# B&R Automation Studio project DeltaTracking (part 2)

#### Cyclic.st - Cyclic code
```iecst
PROGRAM _CYCLIC
	DefineLinks;

	CASE State OF

		/////////////////////////////////////////////////////////////////////////////
		STATE_WAIT:
			/////////////////////////////////////////////////////////////////////////////
			IF  Start THEN
				State := 	STATE_INIT;
			END_IF

		/////////////////////////////////////////////////////////////////////////////
		STATE_INIT:
		////////////////////////////////////////////////////////////////////////////

			IF MpAxConveyor.CommandBusy THEN
				// wait
			ELSIF 	NOT(MpAxConveyor.Active) THEN
				MpAxConveyor.Enable := TRUE;

			ELSIF MpAxConveyor.Error THEN
				MpAxConveyor.ErrorReset := TRUE;

			ELSIF NOT(MpAxConveyor.PowerOn) THEN
				MpAxConveyor.Power := TRUE;

			ELSIF NOT(MpAxConveyor.IsHomed) THEN
				AxParConveyor.Homing.Mode := mcHOMING_DIRECT;
				AxParConveyor.Homing.Position := 0;
				MpAxConveyor.Home := TRUE;

			ELSIF MpAxConveyor.Info.CommunicationReady THEN
				LastProductPosition := MpAxConveyor.Position - ProductGap;
				MC_BR_TrackingFrameDelete_0.Execute := TRUE;
				State := STATE_PRODUCTION;
			END_IF

		//////////////////////////////////////// Frame Handling! + Stat Machine Conveyor///////////////////////////////////////
		STATE_PRODUCTION:
		///////////////////////////////////////////////////////////////////////////////////////////////////////////////////////

			// Move Belt with selected speed
			IF AxParConveyor.Velocity  <> SetVelocity THEN
				// If velocity ist not up to date, update Conveyer Velocity to the Velocity set at the ControlPanel
				MpAxConveyor.Update := TRUE;
			END_IF
			AxParConveyor.Velocity := SetVelocity;
			MpAxConveyor.MoveVelocity := TRUE;

			IF NOT MC_BR_TrackingFrameCreate_0.Busy THEN
				addNewObjects;
			END_IF

			IF MpAxConveyor.Error THEN
				State := STATE_ERROR;

			ELSIF NOT Start THEN
				MpAxConveyor.MoveVelocity := FALSE;

				IF (MpAxConveyor.Error) THEN
					MpAxConveyor.Power := FALSE;
					State := STATE_WAIT;

				ELSIF MpAxConveyor.PowerOn AND NOT(MpAxConveyor.CommandBusy) THEN
					MpAxConveyor.MoveVelocity := FALSE;
					MpAxConveyor.Power := FALSE;

				ELSIF NOT(MpAxConveyor.CommandBusy) THEN
					State := STATE_WAIT;

				END_IF
			END_IF

		///////////////////////////////////////////////////////////////////////////////
		STATE_ERROR:
		///////////////////////////////////////////////////////////////////////////////
			MpAxConveyor.MoveVelocity := FALSE;
			MpAxConveyor.Power := FALSE;

			IF Reset AND MpAxConveyor.Error AND MpAxConveyor.CommandBusy THEN
				MpAxConveyor.ErrorReset := TRUE;

			ELSIF Start AND NOT(MpAxConveyor.Error) AND NOT(MpAxConveyor.CommandBusy) THEN
				State := STATE_WAIT;
			END_IF

	END_CASE

	MpAxConveyor(MpLink := LinkAxis, Parameters := ADR(AxParConveyor), ErrorReset := Reset);
	MC_BR_TrackingFrameCreate_0(TrackingPath := LinkTrackingPath);
	MC_BR_TrackingFrameDelete_0(TrackingPath := LinkTrackingPath);

	IF (MpAxConveyor.Update AND MpAxConveyor.UpdateDone) OR MpAxConveyor.Error THEN
		MpAxConveyor.Update	:= FALSE;
	END_IF

	IF (NOT(MpAxConveyor.MoveActive) AND NOT(MpAxConveyor.CommandBusy)) OR MpAxConveyor.Error THEN
		MpAxConveyor.MoveVelocity := FALSE;
		MpAxConveyor.Update := FALSE;
	END_IF

	IF MpAxConveyor.ErrorReset AND NOT(MpAxConveyor.Error) THEN
		MpAxConveyor.ErrorReset := FALSE;
	END_IF

	IF (MpAxConveyor.Home AND MpAxConveyor.IsHomed) OR MpAxConveyor.Error THEN
		MpAxConveyor.Home := FALSE;
	END_IF

	MC_BR_TrackingFrameCreate_0.Execute	:= FALSE;
	MC_BR_TrackingFrameDelete_0.Execute := FALSE;

END_PROGRAM
```

#### Exit.st - Exit code
```iecst
PROGRAM _EXIT

END_PROGRAM
```

#### DeviceActions.st
```iecst
ACTION addNewObjects:

	// overflow handling
	IF MpAxConveyor.Position < LastProductPosition THEN
		LastProductPosition := LastProductPosition - Period;
	END_IF

	IF MpAxConveyor.Position <  LastProductPosition	+ ProductGap THEN
		RETURN;
	END_IF

	IF Multipick THEN
		MC_BR_TrackingFrameCreate_0.Parameters.Translation.Y := 80 - UDINT_TO_LREAL(createCnt MOD 2) * 160;
		createCnt := createCnt + 1;

		IF createCnt MOD 2 = 0 THEN
			LastProductPosition := MpAxConveyor.Position;
		END_IF

	ELSE
		IF RandomCreation THEN
			MC_BR_TrackingFrameCreate_0.Parameters.Translation.Y := (UINT_TO_LREAL((TIM_musec()*10) MOD 160) - 80);
			MC_BR_TrackingFrameCreate_0.Parameters.Orientation.Angle3 := (UINT_TO_LREAL((TIM_musec()*10) MOD 178)-89);
		ELSE
			MC_BR_TrackingFrameCreate_0.Parameters.Translation.Y := 0;
			MC_BR_TrackingFrameCreate_0.Parameters.Orientation.Angle3 := 0;
		END_IF
		LastProductPosition := MpAxConveyor.Position;
	END_IF

	// simulate two diffent product types
	MC_BR_TrackingFrameCreate_0.Parameters.Attribute := 2#0001;
	IF (TIM_ticks() MOD 2) = 1 THEN
		MC_BR_TrackingFrameCreate_0.Parameters.Attribute := 2#0011;
	END_IF;

	// Add frame in the buffer
	MC_BR_TrackingFrameCreate_0.Parameters.LatchedPath.Position := MpAxConveyor.Position;
	MC_BR_TrackingFrameCreate_0.Execute	:= TRUE;

END_ACTION
```

#### DefineLinks.st
```iecst
ACTION DefineLinks:
	LinkTrackingPath := ADR(gTrackingPathConveyor_1);
	LinkAxis := ADR(gAxis_Conveyor_1);
	Period := 100000.0;

	Reset := ControlPanel.Input.Reset;
	Start :=
		(ControlPanel.Input.StartMultipick OR
		ControlPanel.Input.StartPickNPlace OR
		ControlPanel.Input.StartPlaceWithConditionalStop OR
		ControlPanel.Input.StartPrePalletizing OR
		ControlPanel.Input.StartSorting OR
		ControlPanel.Input.StartMultipickRandom);

	Multipick := ControlPanel.Input.StartMultipick;
	ProductGap := ControlPanel.Input.ProductGap;
	SetVelocity := ControlPanel.Input.VelocityProduction;
	RandomCreation := ControlPanel.Input.StartMultipickRandom;

END_ACTION
```

### Program Logical/Conveyor/APP_Conveyor2 (IEC)

- Cyclic.st (reference to Logical/Conveyor/APP_Conveyor1/Cyclic.st)

- DeviceActions.st (reference to Logical/Conveyor/APP_Conveyor1/DeviceActions.st)

- Exit.st (reference to Logical/Conveyor/APP_Conveyor1/Exit.st)

- Init.st (reference to Logical/Conveyor/APP_Conveyor1/Init.st)

- Variables.var (reference to Logical/Conveyor/APP_Conveyor1/Variables.var)

#### DefineLinks.st
```iecst
ACTION DefineLinks:
	LinkTrackingPath := ADR(gTrackingPathConveyor_2);
	LinkAxis := ADR(gAxis_Conveyor_2);
	Period := 100000.0;

	Reset := ControlPanel.Input.Reset;
	Start :=
		(ControlPanel.Input.StartMultipick OR
		ControlPanel.Input.StartPickNPlace OR
		ControlPanel.Input.StartPlaceWithConditionalStop OR
		ControlPanel.Input.StartPrePalletizing OR
		ControlPanel.Input.StartSorting OR
		ControlPanel.Input.StartMultipickRandom);

	Multipick := ControlPanel.Input.StartMultipick;
	ProductGap := ControlPanel.Input.ProductGap;
	SetVelocity := ControlPanel.Input.VelocityProduction;
	RandomCreation := ControlPanel.Input.StartMultipickRandom;

END_ACTION
```

### Robot.typ
```iecst
TYPE
	RobotStatesEnum :
		( (*State of the robot*)
		ROBOT_WAIT,
		ROBOT_RESET,
		ROBOT_POWER,
		ROBOT_HOME,
		ROBOT_MOVE,
		ROBOT_PRODUCTION,
		ROBOT_ERROR
		);
END_TYPE
```

### Program Logical/Robots/APP_Robot1 (IEC) - Delta1

#### CommonVars.var - Local variables
```iecst
(*
Link handling*)
VAR
	NameAxesGroup : STRING[250]; (*Name of axGroup to find position in object hierachy*)
	LinkAxesGroup : UDINT; (*Link to delta*)
	NameTrackingPath : STRING[250];
	LinkAxisTrackingPath : UDINT;
	LinkTrackingPath : UDINT;
END_VAR
(*
Robot Interface Definition*)
VAR
	MC_BR_GroupStop_X : MC_GroupStop; (*Group object to home axis group*)
	MC_BR_GroupHome_X : MC_BR_GroupHome_15; (*Group object to home axis group*)
	MC_GroupReset_X : MC_GroupReset; (*Group object to home axis group*)
	MC_BR_GroupPower_X : MC_BR_GroupPower; (*Group object to home axis group*)
	MC_BR_GroupReadInfo_X : MC_BR_GroupReadInfo; (*Group object to home axis group*)
	MC_BR_MoveProgram_X : MC_BR_MoveProgram; (*Group object to home axis group*)
	MC_BR_ConditionalStop_0 : MC_BR_ConditionalStop;
	MC_BR_TrackingStatus_PathGen_X : MC_BR_TrackingStatus_PathGen;
	MC_BR_PathInfo_0 : MC_BR_PathInfo;
	MC_BR_GroupReadCyclicPosition_X : MC_BR_GroupReadCyclicPosition_15;
END_VAR
(*
Variables used handling objects and reading informations about the robot*)
VAR
	MC_BR_GetCoordSystemIdent_X : MC_BR_GetCoordSystemIdent;
	MC_BR_TrackingFrameCreate_X : MC_BR_TrackingFrameCreate; (*Tracking Path, read all objects on Path*)
	MC_BR_ReadCyclicPosition_X : MC_BR_ReadCyclicPosition; (*Tracking Path, read all objects on Path*)
END_VAR
(*
Logic*)
VAR
	Reset : BOOL;
	Start : BOOL;
	State : RobotStatesEnum; (*Statemachine*)
END_VAR
(*
Scene Viewer*)
VAR
	GripperClosed : BOOL; (*Scene Viewer*)
	MultigripperClosedPos1 : BOOL; (*Scene Viewer*)
	MultigripperClosedPos2 : BOOL; (*Scene Viewer*)
END_VAR
(*
ST Var*)
VAR
	M16 : BOOL; (*ST Var*)
	M17 : BOOL; (*ST Var*)
	M32 : BOOL; (*ST Var*)
	M33 : BOOL; (*ST Var*)
	M34 : BOOL; (*ST Var*)
	M40 : BOOL; (*ST Var*)
END_VAR
(*
Monitorin Elements*)
VAR
	PickRateWaitForSync : BOOL;
	PickRateCount : UDINT;
	PickRateTimestamp : TIME;
	PickRateTrackingPath : REFERENCE TO McTrackingPathType;
	PickRate : LREAL;
END_VAR
```

#### Init.st - Init code
```iecst
PROGRAM _INIT

	// This action defines the links to the conveyeor and the robot
	DefineLinks;

	MC_BR_PathInfo_0.Enable := TRUE;
	MC_BR_GroupReadInfo_X.Enable := TRUE;
	MC_BR_GroupReadCyclicPosition_X.Enable := TRUE;

	MC_BR_ConditionalStop_0.Enable := TRUE;
	MC_BR_ConditionalStop_0.Identifier := 123;
	MC_BR_ConditionalStop_0.Deactivate := TRUE;
	MC_BR_ConditionalStop_0.Reactivate := FALSE;

	MC_BR_GetCoordSystemIdent_X.CoordSystemName := NameTrackingPath;
	MC_BR_GetCoordSystemIdent_X.Execute := TRUE;
	MC_BR_GetCoordSystemIdent_X();

	MC_BR_ReadCyclicPosition_X.Enable := TRUE;
	MC_BR_ReadCyclicPosition_X.ValueSource := mcVALUE_ACTUAL;

	MC_BR_GroupReadCyclicPosition_X.CoordSystem := MC_BR_GetCoordSystemIdent_X.Ident;

	MC_BR_TrackingStatus_PathGen_X.Enable := TRUE;

END_PROGRAM
```

#### Cyclic.st
```iecst
PROGRAM _CYCLIC
	DefineLinks;

	CASE State OF

		/////////////////////////////////////////////////////////////////////////////
		ROBOT_WAIT:
		/////////////////////////////////////////////////////////////////////////////
			IF  Start THEN
				State := ROBOT_RESET;
			END_IF
			MC_BR_GroupPower_X.Enable := FALSE;
			MultigripperClosedPos1 := FALSE;
			MultigripperClosedPos2 := FALSE;
			GripperClosed := FALSE;
			PickRateCount := 0;

		/////////////////////////////////////////////////////////////////////////////
		ROBOT_RESET:
		/////////////////////////////////////////////////////////////////////////////
			MC_GroupReset_X.Execute := TRUE;
			IF MC_GroupReset_X.Done THEN
				State := ROBOT_POWER;
			END_IF

		/////////////////////////////////////////////////////////////////////////////
		ROBOT_POWER:
		/////////////////////////////////////////////////////////////////////////////
			MC_BR_GroupPower_X.Enable := TRUE;
			IF MC_BR_GroupPower_X.Status THEN
				State := ROBOT_HOME;
			END_IF

		/////////////////////////////////////////////////////////////////////////////
		ROBOT_HOME:
		/////////////////////////////////////////////////////////////////////////////
			MC_BR_GroupHome_X.Execute := TRUE;
			IF MC_BR_GroupHome_X.Done THEN
				State := ROBOT_MOVE;
			END_IF

		/////////////////////////////////////////////////////////////////////////////
		ROBOT_MOVE:
		/////////////////////////////////////////////////////////////////////////////
			MC_BR_MoveProgram_X.Execute := TRUE;
			IF MC_BR_MoveProgram_X.Active THEN
				State := ROBOT_PRODUCTION;
			END_IF

		/////////////////////////////////////////////////////////////////////////////
		ROBOT_PRODUCTION:
		/////////////////////////////////////////////////////////////////////////////

			operateGripper;
			updateConditionalStop;
			calcPickRate;

			IF MC_BR_MoveProgram_X.Done THEN
					State := ROBOT_WAIT;
			ELSIF NOT(Start) THEN
				MC_BR_GroupStop_X.Execute := TRUE;
				IF MC_BR_GroupStop_X.Done THEN
					State := ROBOT_WAIT;
				END_IF
			END_IF

		///////////////////////////////////////////////////////////////////////////////
		ROBOT_ERROR:
		///////////////////////////////////////////////////////////////////////////////
			IF Reset THEN
				State := ROBOT_WAIT;
			END_IF

	END_CASE

	IF MC_GroupReset_X.Error OR MC_BR_GroupPower_X.Error OR MC_BR_GroupHome_X.Error OR MC_BR_MoveProgram_X.Error OR MC_BR_GroupReadInfo_X.Error THEN
		State := ROBOT_ERROR;
	END_IF

	MC_BR_GroupReadInfo_X(AxesGroup := LinkAxesGroup);
	MC_GroupReset_X(AxesGroup := LinkAxesGroup);
	MC_BR_GroupPower_X(AxesGroup := LinkAxesGroup);
	MC_BR_GroupHome_X(AxesGroup := LinkAxesGroup);
	MC_BR_MoveProgram_X(AxesGroup := LinkAxesGroup);
	MC_BR_GroupStop_X(AxesGroup := LinkAxesGroup);
	MC_BR_PathInfo_0(AxesGroup := LinkAxesGroup);
	MC_BR_ConditionalStop_0(AxesGroup := LinkAxesGroup);
	MC_BR_GroupReadCyclicPosition_X(AxesGroup := LinkAxesGroup);
	MC_BR_TrackingFrameCreate_X(TrackingPath := LinkTrackingPath);
	MC_BR_ReadCyclicPosition_X(Axis := LinkAxisTrackingPath);
	MC_BR_TrackingStatus_PathGen_X(AxesGroup := LinkAxesGroup);

	MC_GroupReset_X.Execute := FALSE;
	MC_BR_GroupHome_X.Execute := FALSE;
	MC_BR_MoveProgram_X.Execute := FALSE;
	MC_BR_GroupStop_X.Execute := FALSE;
	MC_BR_TrackingFrameCreate_X.Execute := FALSE;

END_PROGRAM
```

#### Exit.st - Exit code
```iecst
PROGRAM _EXIT

END_PROGRAM
```

#### DeviceActions.st
```iecst
// This action operates the Gripper,
ACTION operateGripper:

	IF M16 THEN
		MultigripperClosedPos1 := FALSE;
		GripperClosed := FALSE;
	END_IF
	IF M17 THEN
		MultigripperClosedPos2 := FALSE;
	END_IF
	IF M32 THEN
		GripperClosed := TRUE;
	END_IF
	IF M33 THEN
		MultigripperClosedPos1 := TRUE;
	END_IF
	IF M34 THEN
		MultigripperClosedPos2 := TRUE;
	END_IF

	IF M40 THEN
		MC_BR_TrackingFrameCreate_X.Parameters.Translation.X := MC_BR_GroupReadCyclicPosition_X.CyclicPosition[0];
		MC_BR_TrackingFrameCreate_X.Parameters.Translation.Y := MC_BR_GroupReadCyclicPosition_X.CyclicPosition[1];
		MC_BR_TrackingFrameCreate_X.Parameters.LatchedPath.Position := MC_BR_ReadCyclicPosition_X.CyclicPosition;
		MC_BR_TrackingFrameCreate_X.Parameters.Attribute := 2#0100;
		MC_BR_TrackingFrameCreate_X.Execute := TRUE;
	END_IF

	M16 := FALSE;
	M17 := FALSE;
	M32 := FALSE;
	M33 := FALSE;
	M34 := FALSE;
	M40 := FALSE;
END_ACTION

ACTION updateConditionalStop:

	// interrupt execution every 3 seconds
	IF  ((TIME_TO_INT(clock_ms()) / 1500) MOD 2) = 0 THEN
		MC_BR_ConditionalStop_0.Reactivate := TRUE;
		MC_BR_ConditionalStop_0.Deactivate := FALSE;
	ELSE
		MC_BR_ConditionalStop_0.Deactivate := TRUE;
		MC_BR_ConditionalStop_0.Reactivate := FALSE;
	END_IF

	MC_BR_ConditionalStop_0.Reactivate := MC_BR_ConditionalStop_0.Reactivate AND NOT MC_BR_ConditionalStop_0.Activated;
	MC_BR_ConditionalStop_0.Deactivate := MC_BR_ConditionalStop_0.Deactivate AND MC_BR_ConditionalStop_0.Activated;

END_ACTION

ACTION calcPickRate:
	PickRateTrackingPath ACCESS LinkTrackingPath;
	IF PickRateWaitForSync
		AND MC_BR_TrackingStatus_PathGen_X.TrackingState = mcPATHGEN_TS_SYNCHRONIZED
		AND PickRateTrackingPath.controlif = MC_BR_TrackingStatus_PathGen_X.TrackingAdditionalInfo.TrackedObject.TrackedTrkPath.controlif THEN

		IF PickRateCount = 0 THEN
			PickRateTimestamp := clock_ms();
		ELSE
			PickRate := 60 * (UDINT_TO_LREAL(PickRateCount) / (TIME_TO_LREAL(clock_ms() - PickRateTimestamp) / 1000.0));
		END_IF
		PickRateCount := PickRateCount + 1;

	END_IF
	PickRateWaitForSync := MC_BR_TrackingStatus_PathGen_X.TrackingState = mcPATHGEN_TS_SYNCHRONIZING;
END_ACTION
```

#### DefineLinks.st
```iecst
ACTION DefineLinks:

	// Define Link to the Robot & Conveyor
	NameAxesGroup	:= 'gAxesGroup_D4r1100R_1';
	LinkAxesGroup	:= ADR(gAxesGroup_D4r1100R_1);

	LinkTrackingPath := ADR(gTrackingPathConveyor_1);
	NameTrackingPath := 'gTrackingPathConveyor_1';
	LinkAxisTrackingPath := ADR(gAxis_Conveyor_1);

	Reset := ControlPanel.Input.Reset;
	Start :=
		(ControlPanel.Input.StartMultipick OR
		ControlPanel.Input.StartPickNPlace OR
		ControlPanel.Input.StartPlaceWithConditionalStop OR
		ControlPanel.Input.StartPrePalletizing OR
		ControlPanel.Input.StartSorting OR
		ControlPanel.Input.StartMultipickRandom);

	IF ControlPanel.Input.StartMultipickRandom THEN
		MC_BR_MoveProgram_X.Name := 'MultipickRandom.st';
	END_IF

	IF ControlPanel.Input.StartMultipick THEN
		MC_BR_MoveProgram_X.Name := 'Multipick.st';
	END_IF

	IF ControlPanel.Input.StartPickNPlace THEN
		MC_BR_MoveProgram_X.Name := 'PickNPlace.st';
	END_IF

	IF ControlPanel.Input.StartPlaceWithConditionalStop THEN
		MC_BR_MoveProgram_X.Name := 'PlaceWithConditionalStop.st';
	END_IF

	IF ControlPanel.Input.StartPrePalletizing THEN
		MC_BR_MoveProgram_X.Name := 'PrePalletizing.st';
	END_IF

	IF ControlPanel.Input.StartSorting THEN
		MC_BR_MoveProgram_X.Name := 'Sorting.st';
	END_IF

END_ACTION
```

### Program Logical/Robots/Robot1/APP_Robot1 (IEC) - Delta1

#### CommonVars.var
```iecst
(*
Link handling*)
VAR
	NameAxesGroup : STRING[250]; (*Name of axGroup to find position in object hierachy*)
	LinkAxesGroup : UDINT; (*Link to delta*)
	NameTrackingPath : STRING[250];
	LinkAxisTrackingPath : UDINT;
	LinkTrackingPath : UDINT;
END_VAR
(*
Robot Interface Definition*)
VAR
	MC_BR_GroupStop_X : MC_GroupStop; (*Group object to home axis group*)
	MC_BR_GroupHome_X : MC_BR_GroupHome_15; (*Group object to home axis group*)
	MC_GroupReset_X : MC_GroupReset; (*Group object to home axis group*)
	MC_BR_GroupPower_X : MC_BR_GroupPower; (*Group object to home axis group*)
	MC_BR_GroupReadInfo_X : MC_BR_GroupReadInfo; (*Group object to home axis group*)
	MC_BR_MoveProgram_X : MC_BR_MoveProgram; (*Group object to home axis group*)
	MC_BR_ConditionalStop_0 : MC_BR_ConditionalStop;
	MC_BR_PathInfo_0 : MC_BR_PathInfo;
	MC_BR_GroupReadCyclicPosition_X : MC_BR_GroupReadCyclicPosition_15;
END_VAR
(*
Variables used handling objects and reading informations about the robot*)
VAR
	MC_BR_GetCoordSystemIdent_X : MC_BR_GetCoordSystemIdent;
	MC_BR_TrackingFrameCreate_X : MC_BR_TrackingFrameCreate; (*Tracking Path, read all objects on Path*)
	MC_BR_ReadCyclicPosition_X : MC_BR_ReadCyclicPosition; (*Tracking Path, read all objects on Path*)
END_VAR
(*
Logic*)
VAR
	Reset : REFERENCE TO BOOL;
	Start : REFERENCE TO BOOL;
	State : RobotStatesEnum; (*Statemachine*)
END_VAR
(*
Scene Viewer*)
VAR
	GripperClosed : BOOL; (*Scene Viewer*)
	MultigripperClosedPos1 : BOOL; (*Scene Viewer*)
	MultigripperClosedPos2 : BOOL; (*Scene Viewer*)
END_VAR
(*
ST Var*)
VAR
	M16 : BOOL; (*ST Var*)
	M17 : BOOL; (*ST Var*)
	M32 : BOOL; (*ST Var*)
	M33 : BOOL; (*ST Var*)
	M34 : BOOL; (*ST Var*)
	M40 : BOOL; (*ST Var*)
END_VAR
(*
Monitorin Elements*)
VAR
	IPMonitor : McProgIntIpMonitorType; (*Monitor to get interpreter line*)
END_VAR
```

#### Cyclic.st
```iecst
PROGRAM _CYCLIC
	DefineLinks;

	CASE State OF

		/////////////////////////////////////////////////////////////////////////////
		ROBOT_WAIT:
		/////////////////////////////////////////////////////////////////////////////
			IF  Start THEN
				State := ROBOT_RESET;
			END_IF
			MC_BR_GroupPower_X.Enable := FALSE;
			MultigripperClosedPos1 := FALSE;
			MultigripperClosedPos2 := FALSE;
			GripperClosed := FALSE;

		/////////////////////////////////////////////////////////////////////////////
		ROBOT_RESET:
		/////////////////////////////////////////////////////////////////////////////
			MC_GroupReset_X.Execute := TRUE;
			IF MC_GroupReset_X.Done THEN
				State := ROBOT_POWER;
			END_IF

		/////////////////////////////////////////////////////////////////////////////
		ROBOT_POWER:
		/////////////////////////////////////////////////////////////////////////////
			MC_BR_GroupPower_X.Enable := TRUE;
			IF MC_BR_GroupPower_X.Status THEN
				State := ROBOT_HOME;
			END_IF

		/////////////////////////////////////////////////////////////////////////////
		ROBOT_HOME:
		/////////////////////////////////////////////////////////////////////////////
			MC_BR_GroupHome_X.Execute := TRUE;
			IF MC_BR_GroupHome_X.Done THEN
				State := ROBOT_MOVE;
			END_IF

		/////////////////////////////////////////////////////////////////////////////
		ROBOT_MOVE:
		/////////////////////////////////////////////////////////////////////////////
			MC_BR_MoveProgram_X.Execute := TRUE;
			IF MC_BR_MoveProgram_X.Active THEN
				State := ROBOT_PRODUCTION;
			END_IF

		/////////////////////////////////////////////////////////////////////////////
		ROBOT_PRODUCTION:
		/////////////////////////////////////////////////////////////////////////////

			operateGripper;
			updateConditionalStop;

			IF MC_BR_MoveProgram_X.Done THEN
					State := ROBOT_WAIT;
			ELSIF NOT(Start) THEN
				MC_BR_GroupStop_X.Execute := TRUE;
				IF MC_BR_GroupStop_X.Done THEN
					State := ROBOT_WAIT;
				END_IF
			END_IF

		///////////////////////////////////////////////////////////////////////////////
		ROBOT_ERROR:
		///////////////////////////////////////////////////////////////////////////////
			IF Reset THEN
				State := ROBOT_WAIT;
			END_IF

	END_CASE

	IF MC_GroupReset_X.Error OR MC_BR_GroupPower_X.Error OR MC_BR_GroupHome_X.Error OR MC_BR_MoveProgram_X.Error OR MC_BR_GroupReadInfo_X.Error THEN
		State := ROBOT_ERROR;
	END_IF

	MC_BR_GroupReadInfo_X(AxesGroup := LinkAxesGroup);
	MC_GroupReset_X(AxesGroup := LinkAxesGroup);
	MC_BR_GroupPower_X(AxesGroup := LinkAxesGroup);
	MC_BR_GroupHome_X(AxesGroup := LinkAxesGroup);
	MC_BR_MoveProgram_X(AxesGroup := LinkAxesGroup);
	MC_BR_GroupStop_X(AxesGroup := LinkAxesGroup);
	MC_BR_PathInfo_0(AxesGroup := LinkAxesGroup);
	MC_BR_ConditionalStop_0(AxesGroup := LinkAxesGroup);
	MC_BR_GroupReadCyclicPosition_X(AxesGroup := LinkAxesGroup);
	MC_BR_TrackingFrameCreate_X(TrackingPath := LinkTrackingPath);
	MC_BR_ReadCyclicPosition_X(Axis := LinkAxisTrackingPath);

	MC_GroupReset_X.Execute := FALSE;
	MC_BR_GroupHome_X.Execute := FALSE;
	MC_BR_MoveProgram_X.Execute := FALSE;
	MC_BR_GroupStop_X.Execute := FALSE;
	MC_BR_TrackingFrameCreate_X.Execute := FALSE;

	IF NOT IPMonitor.Handshake THEN
		IPMonitor.Handshake := TRUE;
	END_IF

END_PROGRAM
```

#### DefineLinks.st
```iecst
ACTION DefineLinks:

	// Define Link to the Robot & Conveyor
	NameAxesGroup	:= 'gAxesGroup_D4r1100_1';
	LinkAxesGroup	:= ADR(gAxesGroup_D4r1100_1);

	LinkTrackingPath := ADR(gTrackingPathConveyor_1);
	NameTrackingPath := 'gTrackingPathConveyor_1';
	LinkAxisTrackingPath := ADR(gAxis_Conveyor_1);

	Reset ACCESS ADR(ControlPanel.Input.Reset);
	Start ACCESS ADR(ControlPanel.Input.StartMultipick);
	MC_BR_MoveProgram_X.Name := 'Multipick.st';

	IF ControlPanel.Input.StartPickNPlace THEN
		MC_BR_MoveProgram_X.Name := 'PickNPlace.st';
		Start ACCESS ADR(ControlPanel.Input.StartPickNPlace);
	END_IF

	IF ControlPanel.Input.StartPlaceWithConditionalStop THEN
		MC_BR_MoveProgram_X.Name := 'PlaceWithConditionalStop.st';
		Start ACCESS ADR(ControlPanel.Input.StartPlaceWithConditionalStop);
	END_IF

	IF ControlPanel.Input.StartPrePalletizing THEN
		MC_BR_MoveProgram_X.Name := 'PrePalletizing.st';
		Start ACCESS ADR(ControlPanel.Input.StartPrePalletizing);
	END_IF

	IF ControlPanel.Input.StartSorting THEN
		MC_BR_MoveProgram_X.Name := 'Sorting.st';
		Start ACCESS ADR(ControlPanel.Input.StartSorting);
	END_IF

END_ACTION
```

#### DeviceActions.st
```iecst
// This action operates the Gripper,
ACTION operateGripper:

	IF M16 THEN
		MultigripperClosedPos1 := FALSE;
		GripperClosed := FALSE;
	END_IF
	IF M17 THEN
		MultigripperClosedPos2 := FALSE;
	END_IF
	IF M32 THEN
		GripperClosed := TRUE;
	END_IF
	IF M33 THEN
		MultigripperClosedPos1 := TRUE;
	END_IF
	IF M34 THEN
		MultigripperClosedPos2 := TRUE;
	END_IF

	IF M40 THEN
		MC_BR_TrackingFrameCreate_X.Parameters.Translation.X := MC_BR_GroupReadCyclicPosition_X.CyclicPosition[0];
		MC_BR_TrackingFrameCreate_X.Parameters.Translation.Y := MC_BR_GroupReadCyclicPosition_X.CyclicPosition[1];
		MC_BR_TrackingFrameCreate_X.Parameters.LatchedPath.Position := MC_BR_ReadCyclicPosition_X.CyclicPosition;
		MC_BR_TrackingFrameCreate_X.Parameters.Attribute := 4;
		MC_BR_TrackingFrameCreate_X.Execute := TRUE;
	END_IF

	M8 := FALSE;
	M16 := FALSE;
	M17 := FALSE;
	M32 := FALSE;
	M33 := FALSE;
	M34 := FALSE;
	M40 := FALSE;
END_ACTION

ACTION updateConditionalStop:

	// interrupt execution every 3 seconds
	IF  ((TIME_TO_INT(clock_ms()) / 1500) MOD 2) = 0 THEN
		MC_BR_ConditionalStop_0.Reactivate := TRUE;
		MC_BR_ConditionalStop_0.Deactivate := FALSE;
	ELSE
		MC_BR_ConditionalStop_0.Deactivate := TRUE;
		MC_BR_ConditionalStop_0.Reactivate := FALSE;
	END_IF

	MC_BR_ConditionalStop_0.Reactivate := MC_BR_ConditionalStop_0.Reactivate AND NOT MC_BR_ConditionalStop_0.Activated;
	MC_BR_ConditionalStop_0.Deactivate := MC_BR_ConditionalStop_0.Deactivate AND MC_BR_ConditionalStop_0.Activated;

END_ACTION
```

#### Init.st
```iecst
PROGRAM _INIT

	// This action defines the links to the conveyeor and the robot
	DefineLinks;

	MC_BR_PathInfo_0.Enable := TRUE;
	MC_BR_GroupReadInfo_X.Enable := TRUE;
	MC_BR_GroupReadCyclicPosition_X.Enable := TRUE;

	MC_BR_ConditionalStop_0.Enable := TRUE;
	MC_BR_ConditionalStop_0.Identifier := 123;
	MC_BR_ConditionalStop_0.Deactivate := TRUE;
	MC_BR_ConditionalStop_0.Reactivate := FALSE;

	MC_BR_GetCoordSystemIdent_X.CoordSystemName := NameTrackingPath;
	MC_BR_GetCoordSystemIdent_X.Execute := TRUE;
	MC_BR_GetCoordSystemIdent_X();

	MC_BR_ReadCyclicPosition_X.Enable := TRUE;
	MC_BR_ReadCyclicPosition_X.ValueSource := mcVALUE_ACTUAL;

	MC_BR_GroupReadCyclicPosition_X.CoordSystem := MC_BR_GetCoordSystemIdent_X.Ident;

END_PROGRAM
```

### Global.var
```iecst
VAR
	ControlPanel : ControlPanelType := (Input:=(Reset:=FALSE,VelocityProduction:=300,ProductGap:=500)); (*Machine interface (inputs/outputs)*)
END_VAR
```

### Multipick.st
```iecst
VAR CONSTANT
	UpperZLevel : LREAL := 100.0;	// Gripper up position
	LowerZLevel : LREAL := 0.0;		// Gripper down position
	YProductPos : LREAL := 200;		// position in y coordinate where the product should be placed
END_VAR

VAR
	ParkPos				: McPointType := (Pos:=(X:=	  0, Y:= 0, 			Z:= UpperZLevel));
	SynchPosUp1			: McPointType := (Pos:=(X:=   -25, Y:= 0, 			Z:= UpperZLevel));
	SynchPosUp2			: McPointType := (Pos:=(X:=   25, Y:= 0, 			Z:= UpperZLevel));
	SynchPosDown1		: McPointType := (Pos:=(X:=   -25, Y:= 0, 			Z:= LowerZLevel));
	SynchPosDown2		: McPointType := (Pos:=(X:=   25, Y:= 0, 			Z:= LowerZLevel));
	StaticMoveDown		: McPointType := (Pos:=(X:=	  0, Y:= 0, 			Z:= 0));
	MoveToPark : BOOL 	:= FALSE;

	FrameIn : McTrkFrmIdentType;
	FrameOut : McTrkFrmIdentType;
END_VAR

PROGRAM _MAIN

	// Position init, reset frame in case of restart
	SetPCS(MachineFrame);
	MoveLR(ParkPos);
	WaitEndMove();

	WaitUntil(TrackingFrameSelect(FrameIn,'Infeed'));				    // hold interpreter until a new frame is available
	REPEAT
		MoveToPark := FALSE;

		TrackObjectR(FrameIn, SynchPosUp2, 50, 50);						// track on product
		MoveLR(SynchPosDown2);											// move to the take position
		WaitTime(0.04);													// Wait cause delay of gripper
		SetM(34);														// Scene - remove product from belt, Close the gripper here
		WaitALAP();
		MoveLR(SynchPosUp2);											// move up to change position

		IF TrackingFrameSelect(FrameIn,'Infeed') THEN
			TrackObjectR(FrameIn, SynchPosUp1, 50, 50);					// track on product
			MoveLR(SynchPosDown1);										// move to the take position
			SetM(33);													// Scene - remove product from belt, Close the gripper here
			WaitTime(0.04);												// Wait cause delay of gripper
			MoveLR(SynchPosUp1);										// move up to change position
		END_IF

		TrackStopR(FixedPlace, ParkPos, 50, 50);						// Move to the fixed place Position
		MoveLR(StaticMoveDown);											// move to the take position
		SetM(16);														// open the gripper here
		SetM(17);														// open the gripper here
		WaitTime(0.04);													// Wait cause delay of gripper
		MoveLR(ParkPos);												// move to the take position
		WaitALAP();

		IF NOT TrackingFrameSelect(FrameIn,'Infeed') THEN				// Need to stop, no objects left
			WaitEndMove();												// sync interpreter and program
			WaitUntil(TrackingFrameSelect(FrameIn,'Infeed'));			// select new product
		END_IF

	UNTIL FALSE END_REPEAT;

END_PROGRAM
```

### PickNPlace.st
```iecst
VAR CONSTANT
	UpperZLevel : LREAL := 100.0;	// Gripper up position
	LowerZLevel : LREAL := 0.0;		// Gripper down position
	YProductPos : LREAL := 200;		// position in y coordinate where the product should be placed
END_VAR

VAR
	ParkPos				: McPointType := (Pos:=(X:=-100, Y:=100, 			Z:= UpperZLevel));
	SynchPosUp			: McPointType := (Pos:=(X:=   0, Y:= 0, 			Z:= UpperZLevel));
	SynchPosDown		: McPointType := (Pos:=(X:=   0, Y:= 0, 			Z:= LowerZLevel));

	FrameIn : McTrkFrmIdentType;
	FrameOut : McTrkFrmIdentType;
END_VAR

PROGRAM _MAIN

	// Position init, reset frame in case of restart
	SetPCS(MachineFrame);
	MoveLR(ParkPos);
	WaitEndMove();

	WaitUntil(TrackingFrameSelect(FrameIn,'Infeed'));				// hold interpreter until a new frame is available
	REPEAT

		TrackObjectR(FrameIn, SynchPosUp, 50, 50);					// track on product
		MoveLR(SynchPosDown);										// move to the take position
		WaitTime(0.04);												// Wait cause delay of gripper
		SetM(32);													// Scene - remove product from belt, close gripper
		WaitALAP();													// hold interpreter

		MoveLR(SynchPosUp);											// move up to change frame
		WaitUntil(TrackingFrameSelect(FrameOut,'Outfeed'));			// hold interpeter until place frame has been selected
		TrackObjectR(FrameOut, SynchPosUp, 50, 50);					// move to place position
		MoveLR(SynchPosDown);										// move down on place position
		WaitTime(0.04);												// Wait cause delay of gripper
		SetM(16);													// Scene - place product on belt, open gripper
		WaitALAP();													// hold interpreter
		TrackingFrameSetAttribute(FrameOut, 4);						// Transfer attribute value

		MoveLR(SynchPosUp);											// move up to change frame
		IF NOT TrackingFrameSelect(FrameIn,'Infeed') THEN			// Need to stop, no objects left
			TrackStopR(MachineFrame, ParkPos, 50, 50);				// Move to a static frame
			WaitEndMove();											// sync interpreter and program
			WaitUntil(TrackingFrameSelect(FrameIn,'Infeed'));		// hold interpreter until a new frame is available
		END_IF

	UNTIL FALSE END_REPEAT;

END_PROGRAM
```

### PlaceWithConditionalStop.st
```iecst
VAR CONSTANT
	UpperZLevel : LREAL := 100.0;	// Gripper up position
	LowerZLevel : LREAL := 0.0;		// Gripper down position
	YProductPos : LREAL := 200;		// position in y coordinate where the product should be placed
END_VAR

VAR
	ParkPos				: McPointType := (Pos:=(X:=	  0, Y:= 0, 			Z:= UpperZLevel));
	SynchPosUp			: McPointType := (Pos:=(X:=   0, Y:= 0, 			Z:= UpperZLevel));
	SynchPosDown		: McPointType := (Pos:=(X:=   0, Y:= 0, 			Z:= LowerZLevel));
	StaticMoveDown		: McPointType := (Pos:=(X:=   0, Y:= 0, 			Z:= -100));
	StaticMoveUp		: McPointType := (Pos:=(X:=   0, Y:= 0, 			Z:= 100));

	FrameIn : McTrkFrmIdentType;
	FrameOut : McTrkFrmIdentType;
END_VAR

PROGRAM _MAIN

	// Position init, reset frame in case of restart
	SetPCS(MachineFrame);
	MoveLR(ParkPos);
	WaitEndMove();

	WaitUntil(TrackingFrameSelect(FrameIn,'Infeed'));				// hold interpreter until a new frame is available
	REPEAT

		TrackObjectR(FrameIn, SynchPosUp, 50, 50);					// track on product
		MoveLR(SynchPosDown);										// move to the take position
		// Close the gripper here
		SetM(32);													// Scene - remove product from belt
		WaitTime(0.04);												// Wait until gripper closes
		MoveLR(SynchPosUp);											// move up to change position

		TrackStopR(FixedPlace, ParkPos, 50, 50);					// Move to the fixed place Position
		ConditionalStop(123);										// Stop movement if place position is not valid
		Relative();													// use relative positions
		MoveLR(StaticMoveDown);										// move to the take position
		WaitEndMove();												// wait to go on with interpreter here
		SetM(16);													// open the gripper here
		WaitTime(0.04);												// Wait until gripper opens
		MoveLR(StaticMoveUp);										// move to the take position
		Absolute();

		IF NOT TrackingFrameSelect(FrameIn,'Infeed') THEN			// Need to stop, no objects left
			MoveLR(ParkPos);										// move to static park position
			WaitEndMove();											// sync interpreter and program
			WaitUntil(TrackingFrameSelect(FrameIn,'Infeed'));		// hold interpreter until a new frame is available
		END_IF

	UNTIL FALSE END_REPEAT;

END_PROGRAM
```

### PrePalletizing.st
```iecst
VAR CONSTANT
	UpperZLevel : LREAL := 100.0;	// Gripper up position
	LowerZLevel : LREAL := 0.0;		// Gripper down position
	YProductPos : LREAL := 200;		// position in y coordinate where the product should be placed
END_VAR

VAR
	ParkPos				: McPointType := (Pos:=(X:=-100, Y:=100, 			Z:= UpperZLevel));
	SynchPosUp			: McPointType := (Pos:=(X:=   0, Y:= 0, 			Z:= UpperZLevel));
	SynchPosDown		: McPointType := (Pos:=(X:=   0, Y:= 0, 			Z:= LowerZLevel));
	SynchPosForward		: McPointType := (Pos:=(X:= 100, Y:= 0, 			Z:= LowerZLevel));
	SynchPosSideward	: McPointType := (Pos:=(X:= 100, Y:= 100, 			Z:= LowerZLevel));
	SynchPosUpSideward	: McPointType := (Pos:=(X:= 100, Y:= 100, 			Z:= UpperZLevel));

	FrameIn : McTrkFrmIdentType;
	FrameOut : McTrkFrmIdentType;
END_VAR

PROGRAM _MAIN

	// Position init, reset frame in case of restart
	SetPCS(MachineFrame);
	MoveLR(ParkPos);
	WaitEndMove();

	WaitUntil(TrackingFrameSelect(FrameIn,'Infeed'));				// hold interpreter until a new frame is available
	REPEAT

		TrackObjectR(FrameIn, SynchPosUp, 50, 50);					// track on product
		MoveLR(SynchPosDown);										// move to the take position
		// close the gripper here
		SetM(32);													// Scene - start moving the poduct on the belt
		WaitTime(0.04);												// Wait cause delay of gripper
		WaitALAP();
		TrackingFrameSetAttribute(FrameIn, 0);						// Hide Object

		Feedrate(15000);											// manipulate with reduced feedrate
		MoveL(SynchPosForward);										// move forward on belt
		MoveL(SynchPosSideward);									// move sideward on belt

		SetM(16);													// open the gripper here
		SetM(40);													// Scene - end of moving the product
		WaitTime(0.04);												// Wait cause delay of gripper
		WaitALAP();													// hold interpreter
		MoveLR(SynchPosUpSideward);									// move up to change frame

		IF NOT TrackingFrameSelect(FrameIn,'Infeed') THEN			// Need to stop, no objects left
			TrackStopR(MachineFrame, ParkPos, 50, 50);				// Move to a static frame
			WaitEndMove();											// sync interpreter and program
			WaitUntil(TrackingFrameSelect(FrameIn,'Infeed'));		// hold interpreter until a new frame is available
		END_IF

	UNTIL FALSE END_REPEAT;

END_PROGRAM
```

### Sorting.st
```iecst
VAR CONSTANT
	UpperZLevel : LREAL := 100.0;	// Gripper up position
	LowerZLevel : LREAL := 0.0;		// Gripper down position
	YProductPos : LREAL := 200;		// position in y coordinate where the product should be placed
END_VAR

VAR
	ParkPos				: McPointType := (Pos:=(X:=	  0, Y:= 0, 			Z:= UpperZLevel));
	SynchPosUp			: McPointType := (Pos:=(X:=   0, Y:= 0, 			Z:= UpperZLevel));
	SynchPosDown		: McPointType := (Pos:=(X:=   0, Y:= 0, 			Z:= LowerZLevel));
	StaticMoveDown		: McPointType := (Pos:=(X:=	  0, Y:= 0, 			Z:= 0));
	MoveToPark : BOOL := FALSE;

	FrameIn : McTrkFrmIdentType;
	FrameOut : McTrkFrmIdentType;
END_VAR

PROGRAM _MAIN

	// Position init, reset frame in case of restart
	SetPCS(MachineFrame);
	MoveLR(ParkPos);
	WaitEndMove();

	WaitUntil(TrackingFrameSelect(FrameIn,'Infeed'));				    // hold interpreter until a new frame is available
	REPEAT
		MoveToPark := FALSE;

		TrackObjectR(FrameIn, SynchPosUp, 50, 50);						// track on product
		MoveLR(SynchPosDown);											// move to the take position
		WaitALAP();														// hold interpreter
		// Close the gripper here
		WaitTime(0.04);													// Wait until gripper opens
		SetM(32);														// Scene - remove product from belt
		MoveLR(SynchPosUp);												// move up to change frame

		IF TrackingFrameGetAttribute(FrameIn) = 1 THEN					// sort out objects of type 1
			TrackStopR(FixedPlace, ParkPos, 50, 50);					// Move to the fixed place Position
			MoveLR(StaticMoveDown);										// move to the take position
			WaitTime(0.04);												// Wait until gripper opens
			SetM(16);													// open the gripper here
			MoveLR(ParkPos);											// move to the take position
			WaitALAP();

			IF NOT TrackingFrameSelect(FrameIn,'Infeed') THEN				// Need to stop, no objects left
				MoveToPark := TRUE;										// force park position
			END_IF

		ELSE

			WaitUntil(TrackingFrameSelect(FrameOut,'Outfeed'));			// hold interpeter until place frame has been selected
			TrackObjectR(FrameOut, SynchPosUp, 50, 50);	// move to place position
			MoveLR(SynchPosDown);										// move down on place position

			SetM(16);													// Scene - place product on belt, Open the gripper here
			WaitTime(0.04);												// Wait until gripper opens
			MoveLR(SynchPosUp);											// move up to change frame
			WaitALAP();													// hold interpreter
			TrackingFrameSetAttribute(FrameOut, 4);						// Transfer attribute value

			IF NOT TrackingFrameSelect(FrameIn,'Infeed') THEN			// Need to stop, no objects left
				TrackStopR(MachineFrame, ParkPos, 50, 50);				// Move to a static frame
				MoveToPark := TRUE;										// force park position
			END_IF

		END_IF

		IF MoveToPark THEN
			MoveLR(ParkPos);											// move to static park position
			WaitEndMove();												// sync interpreter and program
			WaitUntilSync(TrackingFrameSelect(FrameIn,'Infeed'));		// hold interpreter until a new frame is available
		END_IF

	UNTIL FALSE END_REPEAT;

END_PROGRAM
```

### MultipickRandom.st
```iecst
VAR CONSTANT
	UpperZLevel : LREAL := 5.0;		// Gripper up position
	LowerZLevel : LREAL := 0.0;		// Gripper down position
	YProductPos : LREAL := 200;		// position in y coordinate where the product should be placed
END_VAR

VAR
	ParkPos				: McPointType := (Pos:=(X:=	  0, Y:= 0, 			Z:= UpperZLevel));
	SynchPosUp1			: McPointType := (Pos:=(X:=   -25, Y:= 0, 			Z:= UpperZLevel));
	SynchPosUp2			: McPointType := (Pos:=(X:=   25, Y:= 0, 			Z:= UpperZLevel));
	SynchPosDown1		: McPointType := (Pos:=(X:=   -25, Y:= 0, 			Z:= LowerZLevel));
	SynchPosDown2		: McPointType := (Pos:=(X:=   25, Y:= 0, 			Z:= LowerZLevel));
	StaticMoveDown		: McPointType := (Pos:=(X:=	  0, Y:= 0, 			Z:= 0));
	FrameIn : McTrkFrmIdentType;
	FrameOut : McTrkFrmIdentType;
END_VAR

PROGRAM _MAIN

	// Position init, reset frame in case of restart
	SetPCS(MachineFrame);
	MoveLR(ParkPos);
	WaitEndMove();

	WaitUntil(TrackingFrameSelect(FrameIn,'Infeed'));				    // hold interpreter until a new frame is available
	REPEAT
		TrackObjectR(FrameIn, SynchPosUp2, 50, 50);						// track on product
		MoveLR(SynchPosDown2);											// move to the take position
		SetM(34);														// Scene - remove product from belt, Close the gripper here
		WaitTime(0.04);													// Wait cause delay of gripper
		WaitALAP();
		MoveLR(SynchPosUp2);											// move up to change position

		IF TrackingFrameSelect(FrameIn,'Infeed') THEN
			TrackObjectR(FrameIn, SynchPosUp1, 50, 50);					// track on product
			MoveLR(SynchPosDown1);										// move to the take position
			SetM(33);													// Scene - remove product from belt, Close the gripper here
			WaitTime(0.04);												// Wait cause delay of gripper
			MoveLR(SynchPosUp1);										// move up to change position
		END_IF

		TrackStopR(MachineFrame, ParkPos, 50, 50);						// Move to the fixed place Position
		MoveLR(StaticMoveDown);											// move to the take position
		SetM(16);														// open the gripper here
		SetM(17);														// open the gripper here
		WaitTime(0.04);													// Wait cause delay of gripper
		Feedrate(20000);
		MoveL(ParkPos);													// move to the take position
		WaitALAP();

		IF NOT TrackingFrameSelect(FrameIn,'Infeed') THEN				// Need to stop, no objects left
			WaitEndMove();												// sync interpreter and program
			WaitUntil(TrackingFrameSelect(FrameIn,'Infeed'));			// select new product
		END_IF

	UNTIL FALSE END_REPEAT;

END_PROGRAM
```

### MachineInterface.typ - not listed in the package file held
```iecst
TYPE
	ControlPanelInputs : 	STRUCT  (*Command Buttons*)
		StartSorting : BOOL; (*Run a sorting program*)
		StartPrePalletizing : BOOL; (*Run a pre palleticing application demo*)
		StartPickNPlace : BOOL; (*Run a pick and place application demo*)
		StartPlaceWithConditionalStop : BOOL; (*Rund a place position with conditional stop*)
		StartMultipick : BOOL; (*Rund a multipick application demo*)
		Reset : BOOL; (*Stop Execute*)
		VelocityProduction : REAL; (*Velocity for production [ppm]*)
		ProductGap : REAL; (*Length of the product [mm]*)
		DeletePosition : REAL; (*Position where objects are deleted*)
	END_STRUCT;
	ControlPanelType : 	STRUCT  (*Control Panel*)
		Input : ControlPanelInputs; (*Buttons *)
	END_STRUCT;
END_TYPE
```

### MachineInterface.var - not listed in the package file held
```iecst
(*Defines*)
VAR CONSTANT
	MAX_TRACKING_FRAMES : USINT := 200; (*Number of supported objects on the tracking frame*)
	NUM_DEVICES : DINT := 2; (*Number of devices (Robots + Axis)*)
END_VAR
(*Stores the Devices Conveyor & Robot 1*)
VAR CONSTANT
	DEVICES_ARRAY : INT := NUM_DEVICES-1; (*Size of devices array*)
END_VAR
(*Internal states*)
VAR
	ControlPanel : ControlPanelType := (Input:=(Reset:=FALSE,VelocityProduction:=300,ProductGap:=500)); (*Machine interface (inputs/outputs)*)
END_VAR
```

Listed in the project but not available here: Logical/GeneralTexts
